(* IEC 61131-3 sources: CodesysTest/alpha/export/FBs/Components/Bag Delivery/FB_BagDelivery.pou/InPosition.prop, 1 file *)

(* ---- Get.pm.st ---- *)
(*#-#-#-#-#-#-#-#-#-#---Declaration---#-#-#-#-#-#-#-#-#-#-#-#-#*)

VAR
END_VAR
(*#-#-#-#-#-#-#-#-#-#---Implementation---#-#-#-#-#-#-#-#-#-#-#-#-#*)

IF _interconnect = BAG_DELIVERY_IC.EIP THEN
	InPosition := bagFeedMasterMotor.InPosition AND bagFeedRearMotor.InPosition;
ELSE
	InPosition := bagFeedMasterMotor.InPosition;
END_IF
